// TwinCAT 3 PLC project PLC_Eksam2020ET_KEP
// ProgramVersion: 3.1.4023.0
// libraries:
//   Tc2_MC2, * (Beckhoff Automation GmbH)
//   Tc2_Standard, * (Beckhoff Automation GmbH)
//   Tc2_System, * (Beckhoff Automation GmbH)
//   Tc2_Utilities, * (Beckhoff Automation GmbH)
//   Tc3_Module, * (Beckhoff Automation GmbH)
//   SysTime,3.5.9.0,System
// project tree:
//   / Class Diagram.TcCD (not stored), GlobalTextList.TcGTLO, PlcTask.TcTTO, Visualization Manager.TcVMO (not stored)
//   GVLs/ FIO.TcGVL
//   POUs/ HMI.TcPOU, MAIN.TcPOU, P_5MovingToStack.TcPOU, P_3Pack.TcPOU, P_2PickUP.TcPOU, P_4Packing.TcPOU, P_6Stack.TcPOU, P_1Start.TcPOU
//   VISUs/ Visualization_Pos.TcVIS, Visualization_Start_Screen.TcVIS

CONFIGURATION PLC_Eksam2020ET_KEP
    RESOURCE PLC ON TwinCAT3
        TASK PlcTask(INTERVAL := T#10ms, PRIORITY := 20);
        PROGRAM MAIN WITH PlcTask : MAIN;
    END_RESOURCE
END_CONFIGURATION

// ---- GVLs/FIO.TcGVL
{attribute 'qualified_only'}
VAR_GLOBAL
	//SENSORS:


//Bool

bFACTORYRunning: BOOL;
bFACTORYPaused: BOOL;
bFACTORYReset1: BOOL;
bUnknown1: BOOL;
bUnknown2: BOOL;
bPP_ItemDetected: BOOL;
bPP_MovingX: BOOL;
bPP_MovingZ: BOOL;
bPP_BaseDetected: BOOL;
bPP_BaseClamped: BOOL;
bPP_PosLimitBase: BOOL;
bPP_LidClamped: BOOL;
bPP_PosLimitLid: BOOL;
bPP_PartLeaving: BOOL;
bPP_LidDetected: BOOL;
bEbStart: BOOL;
bEbReset: BOOL;
bEbStop: BOOL;
bEbES: BOOL;
bEbManual: BOOL;
bEbAuto: BOOL;
bSC_AtLeft: BOOL;
bInPaMovingXY: BOOL;
bInPaMovinZ: BOOL;
bInPaPosLimit: BOOL;
bInPaBoxDetected: BOOL;
bSC_AtMiddle: BOOL;
bSC_AtRight: BOOL;
bOutPaMovingXY: BOOL;
bOutPaMovingZ: BOOL;
bOutPaPosLimit: BOOL;
bOutPaBoxDetected: BOOL;
bSC_MovingZ: BOOL;
bSC_MovingX: BOOL;
bScAtLoad: BOOL;
bInPaSensBlue: BOOL;
bInPaSensGreen: BOOL;
bInPaSensMetal: BOOL;
bOutPaSens: BOOL;
bSsSensConv1: BOOL;
bSsSensConv2: BOOL;
bSsSensConv3: BOOL;
bPP_BaseSens: BOOL;


//Float

rFACTORYTimeScale: REAL;
rInPaPosY: LREAL;
rInPaPosZ: LREAL;
rInPaPosX: LREAL;
rOutPaPosY: REAL;
rOutPaPosZ: REAL;
rOutPaPosX: REAL;


//Int

iInVision: INT;
iRfidW_ReadData: INT;
iRfidW_CmdId: INT;
iRfidW_Status: INT;
iRfidR_ReadData: INT;
iRfidR_CmdId: INT;
iRfidR_Status: INT;

//ACTUATORS:

//Bool

bFACTORYRun: BOOL;
bFACTORYPause: BOOL;
bFACTORYReset2: BOOL;
bUnknown3: BOOL;
bUnknown4: BOOL;
bUnknown5: BOOL;
bUnknown6: BOOL;
bPP_Grab: BOOL;
bPP_MoveX: BOOL;
bPP_MoveZ: BOOL;
bInEmitBase: BOOL;
bPP_ConvLid: BOOL;
bPP_BaseClamp: BOOL;
bPP_PosRais_Base: BOOL;
bPP_LidClamp: BOOL;
bPP_PosRaise_Lid: BOOL;
bEbStartLight: BOOL;
bEbResetLight: BOOL;
bEbStopLight: BOOL;
bScConv1: BOOL;
bInConvGreen: BOOL;
bInConvMetal: BOOL;
bInConvSorting: BOOL;
bInConvBlue: BOOL;
bInPaGrab: BOOL;
bInPaToolRot: BOOL;
bSC_Left: BOOL;
bSC_Right: BOOL;
bSC_Lift: BOOL;
bOutPaGrab: BOOL;
bOutPaToolRot: BOOL;
bScConv2: BOOL;
bScLoadingConv: BOOL;
bInEmitMetalLid: BOOL;
bInEmitGreenLid: BOOL;
bInEmitBlueLid: BOOL;
bPP_ConvOut: BOOL;
bScEmitPallet: BOOL;
bRollerStopOut: BOOL;
bScConv3: BOOL;
bRfidW_ExeCmd: BOOL;
bRfidR_ExeCmd: BOOL;
bPP_ConvBase2: BOOL;
bPP_ConvBase1: BOOL;


//Float

rInPaMoveY: REAL;
rInPaMoveZ: REAL;
rInPaMoveX: REAL;
rOutPaMoveY: REAL;
rOutPaMoveZ: REAL;
rOutPaMoveX: REAL;

//Int

iFACTORYCameraPosition: INT;
iEbCounter: INT;
iSC_TargetPos: INT;
iRfidW_MemIndex: INT;
iRfidW_WriteData: INT;
iRfidW_Cmd: INT;
iRfidR_MemIndex: INT;
iRfidR_WriteData: INT;
iRfidR_Cmd: INT;
END_VAR

// ---- POUs/MAIN.TcPOU
PROGRAM MAIN
VAR
	
END_VAR

//In Main we just run all our program for pick and place stack mashine. 
//As you can see we have 6 program and a HMI program for our mashine. 

P_1Start();
P_2PickUP();
P_3Pack();
P_4Packing();
P_5MovingToStack();
P_6Stack();
HMI();

END_PROGRAM

// ---- POUs/P_1Start.TcPOU
PROGRAM P_1Start
VAR
	nState: INT;
	
END_VAR

VAR CONSTANT
	//Here we define our constant where we want the different positon to be. This is instead of making steps you can call this fixed steps.
	Standby    : INT := 00;
	Start		:INT := 01;
	atEntry    : INT := 10;
	Moving     : INT := 20;
	MovingStop : INT := 22;
	Waiting    : INT := 30;
	Stopping   : INT := 40;
	Resetting  : INT := 50;
	Estop      : INT := 99;
		
END_VAR

// This is our first program in the program we have made a state mashine  ( Case ... of ) to define what our system should do
// in the different states.



CASE nState OF
	Standby:		
		IF FIO.bEbStart=TRUE THEN
			FIO.bInEmitBase:=TRUE;
			nState:=Start;
		END_IF
		
	Start: // This is where we declair what should happen if a operator have turned the mashine in auto and pressed start.
			FIO.bInEmitBlueLid:=FALSE;
			FIO.bInEmitGreenLid:=FALSE;
			FIO.bInEmitMetalLid:=FALSE;
			
			
		IF FIO.bEbStart=TRUE AND FIO.bEbAuto=TRUE THEN 
			FIO.bInEmitBlueLid:=TRUE;     //Lids will start to spawn 
			FIO.bInEmitGreenLid:=TRUE;
			FIO.bInEmitMetalLid:=TRUE;
			nState:=Moving;
		END_IF

	Moving:	 //when the lids 
		IF FIO.bInEmitBlueLid=TRUE AND FIO.bInPaSensBlue=FALSE THEN
			FIO.bInConvBlue:=TRUE;       
		END_IF
		IF	FIO.bInEmitGreenLid=TRUE AND FIO.bInPaSensGreen=FALSE THEN
			FIO.bInConvGreen:=TRUE;
		END_IF
		IF FIO.bInEmitMetalLid=TRUE AND FIO.bInPaSensMetal=FALSE THEN
			FIO.bInConvMetal:=TRUE;
		END_IF	
			nState:=MovingStop;
			
	MovingStop:		
	 	IF FIO.bInPaSensBlue=TRUE THEN  
			FIO.bInConvBlue:=FALSE;
		END_IF
		IF FIO.bInPaSensGreen=TRUE THEN	
			FIO.bInConvGreen:=FALSE;
		END_IF	
		IF FIO.bInPaSensMetal=TRUE THEN	
			FIO.bInConvMetal:=FALSE;
		END_IF		
			nState := Waiting;			

		
//----------------------------------------------------------------------------//
	Waiting:
			nState:=Moving;
		
//----------------------------------------------------------------------------//
	Stopping:   //when stop is pressed we move into this statement the stop light turn on / This is also the state we start in when we turn on the PLC /System
		IF FIO.bEbStop = FALSE THEN
			FIO.bEbStopLight:=TRUE;
			FIO.bInEmitBase:=FALSE;
		ELSIF FIO.bEbReset=TRUE THEN
			FIO.bEbStopLight:=FALSE;
			nState:=Standby;	
		END_IF
//----------------------------------------------------------------------------//
			
			
		
//----------------------------------------------------------------------------// 			
	ELSE
			nState:=9999;				
END_CASE

IF NOT FIO.bEbStop THEN  
		nState:=Stopping;	
END_IF

END_PROGRAM

// ---- POUs/P_2PickUP.TcPOU
PROGRAM P_2PickUP
VAR
	nState: INT;
	
	//Vision Color for Lid
	Blue:	INT:=3;
	Green:	INT:=6;
	Metal:	INT:=9;
	
	//Timers for the different state to happen. It is good to put in timers so the machinery have time to do the different
	// state before it moves on to the next state else everything will happen really fast.
	fbTimerMoving : TON;	// Timer in the moving state so the XYZ arm have time to process before moving till next state.
	fbTimerPickUP : TON;	 // 
	fbTimerGrab : TON;
	fbTimerGrab2 : TON;
	fbTimerDrop : TON;
	fbTimerMovingLid : TON;
	fbTimerWaiting : TON;
END_VAR

VAR CONSTANT
	//This is the Constant Variables that we use to for the different state in our Case OF Statement.
	Standby: 		INT:=00;
	Start:			INT:=01;
	ReadVision: 	INT:=02;
	atEntry: 		INT:=10;
	Moving: 		INT:=20;
	PickUP:			INT:=21;
	PickUP2: 		INT:=22;
	Grab: 			INT:=23;
	Grab2: 			INT:=24;
	Drop: 			INT:=25;
	MovingLid: 		INT:=26;
	MovingLid2: 	INT:=27;
	MovingStop: 	INT:=29;
	Waiting: 		INT:=30;
	Stopping: 		INT:=40;
	Resetting: 		INT:=50;
	Estop:			INT:=99;
END_VAR

// This is our second program where we emit a base and let the vision cam tell us which color the base is so the first XYZ arm can pick up the lid and send if 
// to pack.


CASE nState OF 
	Standby:	
		IF FIO.bEbStart=TRUE THEN
			nState:=Start;
		END_IF	
	
	Start: 
			IF FIO.bInPaSensBlue AND FIO.bInPaSensGreen AND FIO.bInPaSensMetal THEN
				FIO.bInEmitBase:=TRUE;
				nState:=ReadVision;
			END_IF	
			
	ReadVision: //vision cam read the color of the base
				IF FIO.iInVision=Blue THEN
					FIO.rInPaMoveX:=9;			
					nState:=Moving;	
				END_IF
				IF FIO.iInVision=Green THEN
					FIO.rInPaMoveX:=5;					
					nState:=Moving;
				END_IF
				IF FIO.iInVision=Metal THEN 
					FIO.rInPaMoveX:=1;			
					nState:=Moving;
				END_IF
				
	Moving:
		IF FIO.rInPaMoveX=9 OR FIO.rInPaMoveX=5 OR FIO.rInPaMoveX=1 THEN
			FIO.rInPaMoveY:=0.5;
		 fbTimerMoving(IN:=TRUE,PT:=T#1S);
		 IF fbTimerMoving.Q THEN
			fbTimerMoving(IN:=FALSE);
			nState:=PickUP; 
		 END_IF		
		END_IF
	
	PickUP:
		IF FIO.rInPaMoveY=0.5 THEN
			FIO.rInPaMoveZ:=9;
			FIO.bInPaToolRot:=TRUE;
			fbTimerPickUP(IN:=TRUE,PT:=T#1S);
		 IF fbTimerPickUP.Q THEN
			 fbTimerPickUP(IN:=FALSE);
			nState:=Grab; 
		 END_IF	
		END_IF
		
	Grab:
		IF FIO.rInPaMoveZ=9 THEN
			FIO.bInPaGrab:=TRUE;
		fbTimerGrab(IN:=TRUE,PT:=T#1S);
		 IF fbTimerGrab.Q THEN
			fbTimerGrab(IN:=FALSE);
			nState:=Grab2; 
		 END_IF
		END_IF
		
	Grab2:	
		IF FIO.bInPaGrab=TRUE THEN
			FIO.rInPaMoveZ:=5;
			FIO.rInPaMoveY:=8;
			fbTimerGrab2(IN:=TRUE,PT:=T#1S);	
			IF fbTimerGrab2.Q THEN
				fbTimerGrab2(IN:=FALSE);
				nState:=Drop;
		 	END_IF				
		END_IF
	
	Drop:
		IF FIO.bInPaGrab=TRUE THEN
			FIO.rInPaMoveZ:=8.5;
			fbTimerDrop(IN:=TRUE,PT:=T#1S);	
			IF fbTimerDrop.Q THEN
				fbTimerDrop(IN:=FALSE);
				nState:=MovingLid; 
		 	END_IF
		 END_IF
		 
	MovingLid:				
			IF FIO.rInPaMoveZ=8.5 THEN
				FIO.bInPaGrab:=FALSE;
			END_IF
				fbTimerMovingLid(IN:=TRUE,PT:=T#1S);	
			IF fbTimerMovingLid.Q THEN
				fbTimerMovingLid(IN:=FALSE);
				nState:=MovingLid2; 
		 	END_IF
			
	MovingLid2:		
			IF FIO.bInPaGrab=FALSE THEN
				FIO.rInPaMoveX:=0;
				FIO.rInPaMoveY:=0;
				FIO.rInPaMoveZ:=0;
				FIO.bInPaToolRot:=FALSE;
				FIO.bInConvSorting:=TRUE;
				nState:=waiting; 	
			END_IF
//----------------------------------------------------------------------------//
	Waiting:
			IF FIO.bPP_LidClamp=TRUE THEN
			fbTimerWaiting(IN:=TRUE,PT:=T#1S);	
			IF fbTimerWaiting.Q THEN
				fbTimerWaiting(IN:=FALSE); 
				nState:=Start;
			END_IF
			END_IF
//----------------------------------------------------------------------------//

		

	
	Stopping:
		IF FIO.bEbStop = FALSE THEN
			FIO.bEbStopLight:=TRUE;
		ELSIF FIO.bEbReset=TRUE THEN
				FIO.bEbStopLight:=FALSE;	
			nState:=Standby;	
		END_IF	

//----------------------------------------------------------------------------// 
	ELSE
		nState:=9999;	
END_CASE

IF NOT FIO.bEbStop THEN
		nState:=Stopping;	
END_IF

END_PROGRAM

// ---- POUs/P_3Pack.TcPOU
PROGRAM P_3Pack
VAR
	nState: INT;
	
	fbTimerConvs: TON;
	fbTimerPickUP: TON;
	fbTimerGrab: TON;
	fbMyTimer4: TON;
	fbMyTimer5: TON;
	fbMyTimer6: TON;
	fbMyTimer7 : TON;
	fbMyTimer8 : TON;
	fbMyTimer9 : TON;
	F_TRIGLid:F_TRIG;
END_VAR

VAR CONSTANT
	Standby: 	INT:=00;
	Start:		INT:=01;
	atEntry: 	INT:=10;
	Moving: 	INT:=20;
	MovingStopLidClamp: INT:=21;
	MovingStopBase: 	INT:=22;
	PickUP: 	INT:=23;
	PickUP2: 	INT:=24;
	Grab: 		INT:=25;
	Grab2: 		INT:=26;
	Drop: 		INT:=27;
	Moving2: 	INT:=28;
	MovingPack: INT:=29;
	RaiseBase:	INT:=65;
	StoppingAtSens: INT:= 67;
	Stopping: 	INT:=40;
	Resetting: 	INT:=50;
	Clamp:		INT:=60;
	Waiting: 	INT:=30;
	Estop: 		INT:=99;
	
	
END_VAR

// This is our third program  in this program we put the lid together with the base so it can be a box.


F_TRIGLid(CLK:=FIO.bPP_LidDetected);  //trigger for the sense at the lid pack

CASE nState OF
	Standby: 
		nState:=Start;
 
	Start:    
		IF FIO.bInConvSorting=TRUE THEN
			FIO.bPP_ConvBase1:=TRUE;
			FIO.bPP_ConvBase2:=TRUE;
			FIO.bPP_ConvLid:=TRUE;
			fbTimerConvs(IN:=TRUE,PT:=T#1S);
			IF fbTimerConvs.Q THEN
			fbTimerConvs(IN:=FALSE); 
			nState:=MovingStopBase;
		END_IF	
	END_IF
	
	MovingStopBase:
			IF FIO.bPP_BaseDetected=TRUE THEN
				FIO.bPP_ConvBase1:=FALSE;						
				nState:=MovingStopLidClamp;			
			END_IF
	
			
	MovingStopLidClamp:	  // where the clam for lid and base are activated.
		IF F_TRIGLid.Q THEN
			FIO.bPP_LidClamp:=TRUE;
			FIO.bPP_BaseClamp:=TRUE;	
			nState:=PickUP;
		END_IF
		
	PickUP:
		IF FIO.bPP_LidClamp=TRUE AND FIO.bPP_BaseClamp=TRUE THEN
			FIO.bPP_ConvBase2:=FALSE;
			FIO.bInConvSorting:=FALSE;
			FIO.bPP_MoveX:=TRUE;
			fbTimerPickUP(IN:=TRUE,PT:=T#2S);
				IF fbTimerPickUP.Q THEN
					fbTimerPickUP(IN:=FALSE); 
					nState:=Grab;
				END_IF
		END_IF
	
	Grab:
		IF FIO.bPP_MoveX=TRUE THEN
			FIO.bPP_ConvLid:=FALSE;
			FIO.bPP_MoveZ:=TRUE;
			FIO.bPP_Grab:=TRUE;
			fbTimerGrab(IN:=TRUE,PT:=T#2S);
				IF fbTimerGrab.Q THEN
					fbTimerGrab(IN:=FALSE);
					FIO.bPP_LidClamp:=FALSE; 
					nState:=Grab2;
				END_IF
		END_IF

	Grab2:
		IF FIO.bPP_Grab=TRUE THEN
			FIO.bPP_MoveZ:=FALSE;
			fbMyTimer4(IN:=TRUE,PT:=T#2S);
				IF fbMyTimer4.Q THEN
					fbMyTimer4(IN:=FALSE); 
					FIO.bPP_MoveX:=FALSE;
					nState:=Drop;	
				END_IF			
		END_IF	
	
	Drop:
		IF FIO.bPP_MoveX=FALSE THEN
		fbMyTimer5(IN:=TRUE,PT:=T#2S);
			IF fbMyTimer5.Q THEN
				fbMyTimer5(IN:=FALSE); 
				FIO.bPP_MoveZ:=TRUE;
				nState:=Moving2;	
			END_IF	
		END_IF		
	
	Moving2:
		IF FIO.bPP_MovingX=FALSE THEN	
		fbMyTimer6(IN:=TRUE,PT:=T#2S);
			IF fbMyTimer6.Q THEN
				fbMyTimer6(IN:=FALSE);
				FIO.bPP_Grab:=FALSE; 
				nState:=MovingPack;	
			END_IF							
		END_IF
	
	MovingPack:
		IF FIO.bPP_Grab=FALSE THEN
			FIO.bPP_MoveZ:=FALSE;
			FIO.bPP_BaseClamp:=FALSE;
			fbMyTimer7(IN:=TRUE,PT:=T#2S);
			IF fbMyTimer7.Q THEN
				fbMyTimer7(IN:=FALSE);
				nState:=RaiseBase;	
			END_IF	
		END_IF
	
	RaiseBase:
		IF FIO.bPP_MoveZ=FALSE THEN
			FIO.bPP_PosRais_Base:=TRUE;
			FIO.bPP_ConvBase2:=TRUE;
			FIO.bPP_ConvOut:=TRUE;
			fbMyTimer8(IN:=TRUE,PT:=T#2S);
			IF fbMyTimer8.Q THEN
				fbMyTimer8(IN:=FALSE);
				FIO.bPP_PosRais_Base:=FALSE;
				nState:=StoppingAtSens;	
			END_IF	
		END_IF
		
	StoppingAtSens:
		IF FIO.bOutPaSens = TRUE THEN
			FIO.bPP_ConvOut:=FALSE;
			nState:=Waiting;
		END_IF
//----------------------------------------------------------------------------//

	Waiting:
			nState:=Standby;
		
//----------------------------------------------------------------------------//		
		
	ELSE
		nState:=9999;	
END_CASE

END_PROGRAM

// ---- POUs/P_4Packing.TcPOU
PROGRAM P_4Packing
VAR
	nState: INT;
	
	//Timers
	fbTimerGrabX : TON;
	fbTimerGrabY : TON;
	fbTimerGrabZ : TON;
	fbTimerGrab : TON;
	fbTimerLift : TON;
	fbTimerDrop1 : TON;
	fbTimerDrop2 : TON;
	fbTimerMoving2 : TON;
	fbTimerMoving3 : TON;
	fbTimerMovingLoad : TON;
	fbTimerWaiting : TON;
	fbTimerEmitPal: TON;
	
	iCounterTrig: R_trig;
	
END_VAR
VAR CONSTANT
	//Here we define our constant where we want the different positon to be. This is instead of making steps you can call this fixed steps.
	Standby: 	INT:=00;
	GrabX:		INT:=10;
	GrabY:		INT:=11;
	GrabZ:		INT:=12;
	Grab:		INT:=13;
	Lift:		INT:=15;
	Drop1:		INT:=20;
	Drop2:		INT:=21;
	Moving1    : INT := 30;
	Moving2    : INT := 31;
	Moving3    : INT := 32;
	MovingStop : INT := 22;
	AtLoad:		INT:=35;	
	Waiting    : INT := 40;
	Stopping   : INT := 50;
	Resetting  : INT := 60;
	Estop      : INT := 99;
		
END_VAR

// This is our fourth program is where we count the anount of boxes that have been put together  and the second xyz arm will pick up the box 
// and place it on the pallet.

iCounterTrig(CLK:=FIO.bPP_PosRais_Base);  //define a trigger so we can use it to count the amount of boxes that have been put together.  

IF iCounterTrig.Q THEN                    //box counter
	FIO.iEbCounter:=FIO.iEbCounter+1;
END_IF


 
CASE nState OF
	
	Standby:      //the sensor is true when there are a box and a palled will emit 
		IF  FIO.bOutPaSens=TRUE THEN
			FIO.bScEmitPallet:=TRUE;	
			nState:=GrabX;		
		END_IF	
				

	GrabX:		//we move the XYZ arm in the X position 
		IF FIO.bOutPaSens=TRUE THEN    
			FIO.rOutPaMoveX:=4.5;
			fbTimerGrabX(IN:=TRUE,PT:=T#1S);	
			IF fbTimerGrabX.Q THEN
				fbTimerGrabX(IN:=FALSE); 
				nState:=GrabY;
			END_IF	
		END_IF

	GrabY:	//we move the XYZ arm in the Y position 
		IF FIO.rOutPaMoveX=4.5 THEN 
			FIO.rOutPaMoveY:=9.5;
			fbTimerGrabY(IN:=TRUE,PT:=T#1S);	
			IF fbTimerGrabY.Q THEN
				fbTimerGrabY(IN:=FALSE); 
				nState:=GrabZ;
			END_IF	
		END_IF
	
	GrabZ:  //we move the XYZ arm in the Z position 
		IF FIO.rOutPaMoveY=9.5 THEN 
			FIO.rOutPaMoveZ:=8.5;
			FIO.bOutPaToolRot:=TRUE;
			fbTimerGrabZ(IN:=TRUE,PT:=T#2S);	
			IF fbTimerGrabZ.Q THEN
				fbTimerGrabZ(IN:=FALSE); 
				nState:=Grab;
			END_IF				
		END_IF
	
	Grab:   //we here we turn the grab on so it can pick up a box
		IF FIO.bOutPaBoxDetected=TRUE THEN
			FIO.bOutPaGrab:=TRUE;
			fbTimerGrab(IN:=TRUE,PT:=T#1S);
			 IF fbTimerGrab.Q THEN
				fbTimerGrab(IN:=FALSE);
				nState:=Lift; 
		 	END_IF
		END_IF	
		
	Lift:    //here we lift the box
		IF FIO.bOutPaGrab=TRUE THEN
			FIO.rOutPaMoveZ:=0;
			fbTimerLift(IN:=TRUE,PT:=T#1S);
			 IF fbTimerLift.Q THEN
				fbTimerLift(IN:=FALSE);
				nState:=Drop1;
		 	END_IF					
		END_IF	

	Drop1:  // here move in Y axes so it is almost in the middle of the pallet
		IF FIO.rOutPaMoveZ=0 THEN
			FIO.rOutPaMoveY:=1.5;
			fbTimerDrop1(IN:=TRUE,PT:=T#1S);
			 IF fbTimerDrop1.Q THEN
				fbTimerDrop1(IN:=FALSE);
				nState:=Drop2;
		 	END_IF
		END_IF	
		
	Drop2:  //here we move the arm in Z position where we lower the har closer to the pallet and then we drop the box
		IF FIO.bOutPaGrab=TRUE THEN
			FIO.rOutPaMoveZ:=10;
			fbTimerDrop2(IN:=TRUE,PT:=T#1S);
			 IF fbTimerDrop2.Q THEN
				fbTimerDrop2(IN:=FALSE);
				FIO.bOutPaGrab:=FALSE;
				nState:=Waiting;;
		 	END_IF	
		END_IF


		
//----------------------------------------------------------------------------//

	Waiting:
			nState:=Standby;
		
			
		
//----------------------------------------------------------------------------//


	ELSE
		nState:=9999;	
END_CASE

END_PROGRAM

// ---- POUs/P_5MovingToStack.TcPOU
PROGRAM P_5MovingToStack
VAR
	nState: INT;
	
	//Timers
	fbTimerGrabX : TON;
	fbTimerGrabY : TON;
	fbTimerGrabZ : TON;
	fbTimerGrab : TON;
	fbTimerLift : TON;
	fbTimerDrop1 : TON;
	fbTimerDrop2 : TON;
	fbTimerMoving1 : TON;
	fbTimerMoving2 : TON;
	fbTimerMoving3 : TON;
	fbTimerMovingLoad : TON;
	fbTimerWaiting : TON;
	fbTimerEmitPal: TON;
END_VAR
VAR CONSTANT
	Standby: 	INT := 00;
	atEntry: 	INT := 10;
	GrabX:		INT:=10;
	GrabY:		INT:=11;
	GrabZ:		INT:=12;
	Grab:		INT:=13;
	Lift:		INT:=15;
	Drop1:		INT:=20;
	Drop2:		INT:=21;
	Moving1    : INT := 30;
	Moving2    : INT := 31;
	Moving3    : INT := 32;
	MovingStop : INT := 22;
	AtLoad:		INT:=35;	
	Waiting    : INT := 40;
	Stopping   : INT := 50;
	Resetting  : INT := 60;
	Estop      : INT := 9999;
	
	
END_VAR

// This is our fifth program where we make sure to emit a pallet sent the XYZ arn to it's start position. 
// it is also here where we move the pallet with box so it can be stacked in the next program

//we have a If statement when the sensor at the OutPaSens is true then we emit a pallet else we don't.
IF  FIO.bOutPaSens=TRUE THEN    
	FIO.bScEmitPallet:=TRUE;
ELSE 
	FIO.bScEmitPallet:=FALSE;			
END_IF	

CASE nState OF 
	Standby: // we make sure that the grab have stop and there are no box at the OutPaSens then the xyz arm cna move to its home position. 
		IF FIO.bOutPaGrab=FALSE AND FIO.bSsSensConv1=TRUE AND FIO.bOutPaSens=FALSE THEN
			FIO.rOutPaMoveX:=0;
			FIO.rOutPaMoveY:=0;
			FIO.rOutPaMoveZ:=0;
			FIO.bOutPaToolRot:=FALSE;
			fbTimerMoving2(IN:=TRUE,PT:=T#1S);
			IF fbTimerMoving2.Q THEN
				fbTimerMoving2(IN:=FALSE);
				nState:=Moving1;
			END_IF
		END_IF
		
	Moving1:  // if the Sensor at Conveyor1 is True it means there is a pallet  and the grab is false that mean that the box have been delivered 
			IF FIO.bSsSensConv1=TRUE AND FIO.bOutPaGrab=FALSE AND FIO.rOutPaMoveX=0 THEN  
					FIO.bScConv1:=TRUE; //here we start the convayer so the pallet can move 
					nState:=Moving2;
			END_IF

	
	Moving2:  // moving to next conveayer 
		IF FIO.bSsSensConv2=TRUE THEN
			FIO.bScConv2:=TRUE;
			fbTimerMoving2(IN:=TRUE,PT:=T#1S);
			 IF fbTimerMoving2.Q THEN
				fbTimerMoving2(IN:=FALSE);
				FIO.bScConv1:=FALSE;
				nState:=Moving3;
		 	END_IF					 
		END_IF
	
	Moving3: //moving though the last conveyor before it is at the load conveyor. 
		IF FIO.bSsSensConv3=TRUE THEN 
			FIO.bScConv3:=TRUE;
			fbTimerMoving3(IN:=TRUE,PT:=T#1S);
			 IF fbTimerMoving3.Q THEN
				fbTimerMoving3(IN:=FALSE);
				FIO.bScConv2:=FALSE;
				nState:=Waiting;
		 	END_IF						
		END_IF
		
//----------------------------------------------------------------------------//

	Waiting:
			nState:=Standby;
		
//----------------------------------------------------------------------------//		
		
	ELSE 
		nState:=9999; 	
		
END_CASE

END_PROGRAM

// ---- POUs/P_6Stack.TcPOU
PROGRAM P_6Stack
VAR
	nState: INT;
	
	//Timers
	fbTimerMovingLoad: TON;
	fbTimerLift: TON;
	fbTimerToSpace: TON;
	fbTimerPlace: TON;
	fbTimerCounter: TON;
	fbTimerHoming: TON;
	
	
	AtLoadTrig:R_TRIG;		

	//INT
	nCounter         : INT := 0;
END_VAR

VAR CONSTANT
	//Here we define our constant where we want the different positon to be. This is instead of making steps you can call this fixed steps.
	Start		:INT:=00;
	AtLoad		:INT:=01;
	PickUP 		:INT := 02;
	LiftPallet         : INT := 03;
	RetractForksLeft   : INT := 04;
	MovingToSpace      : INT := 05;
	DeliverPart        : INT := 06;
	PlacePallet        : INT := 07;
	RetractRight       : INT := 08;
	Homing             : INT := 09;
	Retry   		   : INT := 10;
	Moving     : INT := 20;
	MovingStop : INT := 22;
	GetPart            : INT := 50;
	GetPartPick        : INT := 51;
	PartPickUp    	   : INT := 52;
	PickUpPart         : INT := 53;
	PartPicked 		   : INT := 54;
	MoveToUnload       : INT := 55;
	UnloadPart 		   : INT := 56;
	PlacePart          : INT := 57;
	Waiting    : INT := 30;	
	Stopping   : INT := 40;
	Resetting  : INT := 60;
	Estop      : INT := 9999;		
END_VAR

// This is our sixth program the stacker robot will pick up the pallet at load and stack them into the different shelf from 1 to 54. 


AtLoadTrig(CLK:=FIO.bScAtLoad);


CASE nState OF
		Start: //Entry of the Palled 
			IF FIO.bScAtLoad=FALSE AND FIO.bScConv3=TRUE THEN
				FIO.bScLoadingConv:=TRUE;                       //turning on the load conveyor
			END_IF
				FIO.iSC_TargetPos := 21474; //This is the value that sends the crane home.
			
			IF AtLoadTrig.Q THEN // counter for the stack robot to know which shelf to put the palled in shelf no = anount of pallet that have been at entry.
			nCounter:=nCounter+1;
			END_IF
			IF FIO.bScAtLoad=TRUE THEN
				nState := AtLoad;
			END_IF
		
		AtLoad:	 // Pallet is at load, the different conveyor will go false when pallet is at load.
		IF FIO.bScAtLoad=TRUE THEN 
			FIO.bScLoadingConv:=FALSE;
			fbTimerMovingLoad(IN:=TRUE,PT:=T#1S);
			IF fbTimerMovingLoad.Q THEN
				fbTimerMovingLoad(IN:=FALSE);
				FIO.bScConv3:=FALSE;
				nState := PickUP;
		 	END_IF						
		END_IF	

	PickUP:  // here we make sure that the the stack robot are at home and there pallet at the load and moving x and z are false before it cna pick up a pallet.
		IF FIO.bScAtLoad=TRUE AND FIO.iSC_TargetPos = 21474 AND FIO.bSC_MovingX=FALSE and FIO.bSC_MovingZ=FALSE THEN
			FIO.bSc_Left := TRUE;
			nState := LiftPallet;
		END_IF
	
	LiftPallet:	 // there the pallet gets picked up	
		IF FIO.bSc_AtLeft=TRUE THEN
			FIO.bSc_Lift:=TRUE;
			fbTimerLift(IN:=TRUE,PT:=T#1S);	
			IF fbTimerLift.Q THEN
				fbTimerLift(IN:=FALSE);
				FIO.bSc_Left :=FALSE; 
				nState := RetractForksLeft;
			END_IF	
		END_IF
	
	RetractForksLeft:  // here er made an extra step to give time for the fock to come back before we move to the next state
			nState:= MovingToSpace;
			
	MovingToSpace:	// here we make sure that the pallet are at mid before the stack robot moves again and we cound which palle 
		IF 	FIO.bSC_AtMiddle=TRUE THEN
			FIO.iSC_TargetPos:=nCounter;    //here we set the pallet count = the target pos which is the space in the shelf
			fbTimerToSpace(IN:=TRUE,PT:=T#2S);	
			IF fbTimerToSpace.Q THEN
				fbTimerToSpace(IN:=FALSE);
				nState := DeliverPart;
			END_IF
		END_IF

	DeliverPart: // here we put pallet into shelf                             
		IF FIO.bSC_MovingX=FALSE THEN
		FIO.bSc_Right := TRUE;                    
		nState := PlacePallet;
		END_IF
		
	PlacePallet:   
		IF FIO.bSc_AtRight=TRUE THEN
			FIO.bSc_Lift:=FALSE;
			fbTimerPlace(IN:=TRUE,PT:=T#1S);	
			IF fbTimerPlace.Q THEN
				fbTimerPlace(IN:=FALSE);
				nState := RetractRight;
			END_IF	
		END_IF

   		RetractRight:   //retract the arm     
		    IF FIO.bSc_Lift=FALSE THEN
				FIO.bSc_Right:=FALSE;
			fbTimerHoming(IN:=TRUE,PT:=T#1S);	
			IF fbTimerHoming.Q THEN
				fbTimerHoming(IN:=FALSE);
				nState := Homing; 		
			END_IF				
		END_IF

	Homing:		//moving to homing
		IF FIO.bSc_AtMiddle=TRUE THEN
			FIO.iSc_TargetPos := 21474;
			nState := Start;	
		END_IF		
		
	ELSE

	nState:=9999;		
	
END_CASE

END_PROGRAM

// ---- POUs/HMI.TcPOU
PROGRAM HMI
VAR

	SpaceOcc1: BOOL;
	
	nState: INT;
	nLastState: INT;
	
	nCounter: INT;
	EmitTrig:R_TRIG;

	Lamp1_Blue: BOOL;
	Lamp1_Green: BOOL;
	Lamp1_Metal: BOOL;	
	Lamp2_Blue: BOOL;
	Lamp2_Green: BOOL;
	Lamp2_Metal: BOOL;
	Lamp3_Blue: BOOL;
	Lamp3_Green: BOOL;
	Lamp3_Metal: BOOL;
	Lamp4_Blue: BOOL;
	Lamp4_Green: BOOL;
	Lamp4_Metal: BOOL;
	Lamp5_Blue: BOOL;
	Lamp5_Green: BOOL;
	Lamp5_Metal: BOOL;
	Lamp6_Blue: BOOL;
	Lamp6_Green: BOOL;
	Lamp6_Metal: BOOL;
	Lamp7_Blue: BOOL;
	Lamp7_Green: BOOL;
	Lamp7_Metal: BOOL;	
	Lamp8_Blue: BOOL;
	Lamp8_Green: BOOL;
	Lamp8_Metal: BOOL;
	Lamp9_Blue: BOOL;
	Lamp9_Green: BOOL;
	Lamp9_Metal: BOOL;
	Lamp10_Blue: BOOL;
	Lamp10_Green: BOOL;
	Lamp10_Metal: BOOL;
	Lamp11_Blue: BOOL;
	Lamp11_Green: BOOL;
	Lamp11_Metal: BOOL;
	Lamp12_Blue: BOOL;
	Lamp12_Green: BOOL;
	Lamp12_Metal: BOOL;
	Lamp13_Blue: BOOL;
	Lamp13_Green: BOOL;
	Lamp13_Metal: BOOL;
	Lamp14_Blue: BOOL;
	Lamp14_Green: BOOL;
	Lamp14_Metal: BOOL;
	Lamp15_Blue: BOOL;
	Lamp15_Green: BOOL;
	Lamp15_Metal: BOOL;
	Lamp16_Blue: BOOL;
	Lamp16_Green: BOOL;
	Lamp16_Metal: BOOL;
	Lamp17_Blue: BOOL;
	Lamp17_Green: BOOL;
	Lamp17_Metal: BOOL;
	Lamp18_Blue: BOOL;
	Lamp18_Green: BOOL;
	Lamp18_Metal: BOOL;
	Lamp19_Blue: BOOL;
	Lamp19_Green: BOOL;
	Lamp19_Metal: BOOL;	
	Lamp20_Blue: BOOL;
	Lamp20_Green: BOOL;
	Lamp20_Metal: BOOL;
	Lamp21_Blue: BOOL;
	Lamp21_Green: BOOL;
	Lamp21_Metal: BOOL;
	Lamp22_Blue: BOOL;
	Lamp22_Green: BOOL;
	Lamp22_Metal: BOOL;
	Lamp23_Blue: BOOL;
	Lamp23_Green: BOOL;
	Lamp23_Metal: BOOL;
	Lamp24_Blue: BOOL;
	Lamp24_Green: BOOL;
	Lamp24_Metal: BOOL;
	Lamp25_Blue: BOOL;
	Lamp25_Green: BOOL;
	Lamp25_Metal: BOOL;
	Lamp26_Blue: BOOL;
	Lamp26_Green: BOOL;
	Lamp26_Metal: BOOL;
	Lamp27_Blue: BOOL;
	Lamp27_Green: BOOL;
	Lamp27_Metal: BOOL;
	Lamp28_Blue: BOOL;
	Lamp28_Green: BOOL;
	Lamp28_Metal: BOOL;
	Lamp29_Blue: BOOL;
	Lamp29_Green: BOOL;
	Lamp29_Metal: BOOL;	
	Lamp30_Blue: BOOL;
	Lamp30_Green: BOOL;
	Lamp30_Metal: BOOL;
	Lamp31_Blue: BOOL;
	Lamp31_Green: BOOL;
	Lamp31_Metal: BOOL;
	Lamp32_Blue: BOOL;
	Lamp32_Green: BOOL;
	Lamp32_Metal: BOOL;
	Lamp33_Blue: BOOL;
	Lamp33_Green: BOOL;
	Lamp33_Metal: BOOL;
	Lamp34_Blue: BOOL;
	Lamp34_Green: BOOL;
	Lamp34_Metal: BOOL;
	Lamp35_Blue: BOOL;
	Lamp35_Green: BOOL;
	Lamp35_Metal: BOOL;
	Lamp36_Blue: BOOL;
	Lamp36_Green: BOOL;
	Lamp36_Metal: BOOL;
	Lamp37_Blue: BOOL;
	Lamp37_Green: BOOL;
	Lamp37_Metal: BOOL;
	Lamp38_Blue: BOOL;
	Lamp38_Green: BOOL;
	Lamp38_Metal: BOOL;
	Lamp39_Blue: BOOL;
	Lamp39_Green: BOOL;
	Lamp39_Metal: BOOL;	
	Lamp40_Blue: BOOL;
	Lamp40_Green: BOOL;
	Lamp40_Metal: BOOL;	
	Lamp41_Blue: BOOL;
	Lamp41_Green: BOOL;
	Lamp41_Metal: BOOL;	
	Lamp42_Blue: BOOL;
	Lamp42_Green: BOOL;
	Lamp42_Metal: BOOL;	
	Lamp43_Blue: BOOL;
	Lamp43_Green: BOOL;
	Lamp43_Metal: BOOL;	
	Lamp44_Blue: BOOL;
	Lamp44_Green: BOOL;
	Lamp44_Metal: BOOL;	
	Lamp45_Blue: BOOL;
	Lamp45_Green: BOOL;
	Lamp45_Metal: BOOL;	
	Lamp46_Blue: BOOL;
	Lamp46_Green: BOOL;
	Lamp46_Metal: BOOL;	
	Lamp47_Blue: BOOL;
	Lamp47_Green: BOOL;
	Lamp47_Metal: BOOL;	
	Lamp48_Blue: BOOL;
	Lamp48_Green: BOOL;
	Lamp48_Metal: BOOL;	
	Lamp49_Blue: BOOL;
	Lamp49_Green: BOOL;
	Lamp49_Metal: BOOL;		
	Lamp50_Blue: BOOL;
	Lamp50_Green: BOOL;
	Lamp50_Metal: BOOL;	
	Lamp51_Blue: BOOL;
	Lamp51_Green: BOOL;
	Lamp51_Metal: BOOL;	
	Lamp52_Blue: BOOL;
	Lamp52_Green: BOOL;
	Lamp52_Metal: BOOL;	
	Lamp53_Blue: BOOL;
	Lamp53_Green: BOOL;
	Lamp53_Metal: BOOL;	
	Lamp54_Blue: BOOL;
	Lamp54_Green: BOOL;
	Lamp54_Metal: BOOL;		



END_VAR

// In this program we setup the link between the stacking shelf with the HMI,
// it is here we set the lamps that will show what color box that are on the shelf
// and what shelf number the boxes are on. 
// It is also here we link the start and stop from HMI, and the auto status. 
// We have not made so you can put the system in auto on the HMI, this is due to safty. 

EmitTrig(CLK:=FIO.bPP_BaseSens);

IF EmitTrig.Q THEN				// This is the counter that are linked with the HIM to se the shelf number the boxes go in.
	nCounter:=nCounter+1;
END_IF


//---------------------------------------------------

IF nCounter = 1 AND FIO.iInVision = 3 THEN   // Linking the self number with the color of the box  throw the vision sencor.
        Lamp1_Blue := TRUE;
END_IF	
IF nCounter = 1 AND FIO.iInVision = 6 THEN  
        Lamp1_Green := TRUE;
END_IF		
IF nCounter = 1 AND FIO.iInVision = 9 THEN
        Lamp1_Metal := TRUE;
END_IF		

//---------------------------------------------------
	
IF nCounter = 2 AND FIO.iInVision = 3 THEN
        Lamp2_Blue := TRUE;
END_IF	
IF nCounter = 2 AND FIO.iInVision = 6 THEN
        Lamp2_Green := TRUE;
END_IF		
IF nCounter = 2 AND FIO.iInVision = 9 THEN
        Lamp2_Metal := TRUE;
END_IF	


//---------------------------------------------------

IF nCounter = 3 AND FIO.iInVision = 3 THEN
        Lamp3_Blue := TRUE;
END_IF	
IF nCounter = 3 AND FIO.iInVision = 6 THEN
        Lamp3_Green := TRUE;
END_IF		
IF nCounter = 3 AND FIO.iInVision = 9 THEN
        Lamp3_Metal := TRUE;
END_IF


//---------------------------------------------------

IF nCounter = 4 AND FIO.iInVision = 3 THEN
        Lamp4_Blue := TRUE;
END_IF	
IF nCounter = 4 AND FIO.iInVision = 6 THEN
        Lamp4_Green := TRUE;
END_IF		
IF nCounter = 4 AND FIO.iInVision = 9 THEN
        Lamp4_Metal := TRUE;
END_IF

//---------------------------------------------------

IF nCounter = 5 AND FIO.iInVision = 3 THEN
        Lamp5_Blue := TRUE;
END_IF	
IF nCounter = 5 AND FIO.iInVision = 6 THEN
        Lamp5_Green := TRUE;
END_IF		
IF nCounter = 5 AND FIO.iInVision = 9 THEN
        Lamp5_Metal := TRUE;
END_IF

//---------------------------------------------------

IF nCounter = 6 AND FIO.iInVision = 3 THEN
        Lamp6_Blue := TRUE;
END_IF	
IF nCounter = 6 AND FIO.iInVision = 6 THEN
        Lamp6_Green := TRUE;
END_IF		
IF nCounter = 6 AND FIO.iInVision = 9 THEN
        Lamp6_Metal := TRUE;
END_IF

//---------------------------------------------------

IF nCounter = 7 AND FIO.iInVision = 3 THEN
        Lamp7_Blue := TRUE;
END_IF	
IF nCounter = 7 AND FIO.iInVision = 6 THEN
        Lamp7_Green := TRUE;
END_IF		
IF nCounter = 7 AND FIO.iInVision = 9 THEN
        Lamp7_Metal := TRUE;
END_IF

//---------------------------------------------------

IF nCounter = 8 AND FIO.iInVision = 3 THEN
        Lamp8_Blue := TRUE;
END_IF	
IF nCounter = 8 AND FIO.iInVision = 6 THEN
        Lamp8_Green := TRUE;
END_IF		
IF nCounter = 8 AND FIO.iInVision = 9 THEN
        Lamp8_Metal := TRUE;
END_IF

//---------------------------------------------------

IF nCounter = 9 AND FIO.iInVision = 3 THEN
        Lamp9_Blue := TRUE;
END_IF	
IF nCounter = 9 AND FIO.iInVision = 6 THEN
        Lamp9_Green := TRUE;
END_IF		
IF nCounter = 9 AND FIO.iInVision = 9 THEN
        Lamp9_Metal := TRUE;
END_IF

//---------------------------------------------------

IF nCounter = 10 AND FIO.iInVision = 3 THEN
        Lamp10_Blue := TRUE;
END_IF	
IF nCounter = 10 AND FIO.iInVision = 6 THEN
        Lamp10_Green := TRUE;
END_IF		
IF nCounter = 10 AND FIO.iInVision = 9 THEN
        Lamp10_Metal := TRUE;
END_IF

//---------------------------------------------------

IF nCounter = 11 AND FIO.iInVision = 3 THEN
        Lamp11_Blue := TRUE;
END_IF	
IF nCounter = 11 AND FIO.iInVision = 6 THEN
        Lamp11_Green := TRUE;
END_IF		
IF nCounter = 11 AND FIO.iInVision = 9 THEN
        Lamp11_Metal := TRUE;
END_IF

//---------------------------------------------------

IF nCounter = 12 AND FIO.iInVision = 3 THEN
        Lamp12_Blue := TRUE;
END_IF	
IF nCounter = 12 AND FIO.iInVision = 6 THEN
        Lamp12_Green := TRUE;
END_IF		
IF nCounter = 12 AND FIO.iInVision = 9 THEN
        Lamp12_Metal := TRUE;
END_IF

//---------------------------------------------------

IF nCounter = 13 AND FIO.iInVision = 3 THEN
        Lamp13_Blue := TRUE;
END_IF	
IF nCounter = 13 AND FIO.iInVision = 6 THEN
        Lamp13_Green := TRUE;
END_IF		
IF nCounter = 13 AND FIO.iInVision = 9 THEN
        Lamp13_Metal := TRUE;
END_IF

//---------------------------------------------------

IF nCounter = 14 AND FIO.iInVision = 3 THEN
        Lamp14_Blue := TRUE;
END_IF	
IF nCounter = 14 AND FIO.iInVision = 6 THEN
        Lamp14_Green := TRUE;
END_IF		
IF nCounter = 14 AND FIO.iInVision = 9 THEN
        Lamp14_Metal := TRUE;
END_IF

//---------------------------------------------------

IF nCounter = 15 AND FIO.iInVision = 3 THEN
        Lamp15_Blue := TRUE;
END_IF	
IF nCounter = 15 AND FIO.iInVision = 6 THEN
        Lamp15_Green := TRUE;
END_IF		
IF nCounter = 15 AND FIO.iInVision = 9 THEN
        Lamp15_Metal := TRUE;
END_IF

//---------------------------------------------------

IF nCounter = 16 AND FIO.iInVision = 3 THEN
        Lamp16_Blue := TRUE;
END_IF	
IF nCounter = 16 AND FIO.iInVision = 6 THEN
        Lamp16_Green := TRUE;
END_IF		
IF nCounter = 16 AND FIO.iInVision = 9 THEN
        Lamp16_Metal := TRUE;
END_IF

//---------------------------------------------------

IF nCounter = 17 AND FIO.iInVision = 3 THEN
        Lamp17_Blue := TRUE;
END_IF	
IF nCounter = 17 AND FIO.iInVision = 6 THEN
        Lamp17_Green := TRUE;
END_IF		
IF nCounter = 17 AND FIO.iInVision = 9 THEN
        Lamp17_Metal := TRUE;
END_IF

//---------------------------------------------------

IF nCounter = 18 AND FIO.iInVision = 3 THEN
        Lamp18_Blue := TRUE;
END_IF	
IF nCounter = 18 AND FIO.iInVision = 6 THEN
        Lamp18_Green := TRUE;
END_IF		
IF nCounter = 18 AND FIO.iInVision = 9 THEN
        Lamp18_Metal := TRUE;
END_IF

//---------------------------------------------------

IF nCounter = 19 AND FIO.iInVision = 3 THEN
        Lamp19_Blue := TRUE;
END_IF	
IF nCounter = 19 AND FIO.iInVision = 6 THEN
        Lamp19_Green := TRUE;
END_IF		
IF nCounter = 19 AND FIO.iInVision = 9 THEN
        Lamp19_Metal := TRUE;
END_IF

//---------------------------------------------------

IF nCounter = 20 AND FIO.iInVision = 3 THEN
        Lamp20_Blue := TRUE;
END_IF	
IF nCounter = 20 AND FIO.iInVision = 6 THEN
        Lamp20_Green := TRUE;
END_IF		
IF nCounter = 20 AND FIO.iInVision = 9 THEN
        Lamp20_Metal := TRUE;
END_IF

//---------------------------------------------------

IF nCounter = 21 AND FIO.iInVision = 3 THEN
        Lamp21_Blue := TRUE;
END_IF	
IF nCounter = 21 AND FIO.iInVision = 6 THEN
        Lamp21_Green := TRUE;
END_IF		
IF nCounter = 21 AND FIO.iInVision = 9 THEN
        Lamp21_Metal := TRUE;
END_IF

//---------------------------------------------------

IF nCounter = 22 AND FIO.iInVision = 3 THEN
        Lamp22_Blue := TRUE;
END_IF	
IF nCounter = 22 AND FIO.iInVision = 6 THEN
        Lamp22_Green := TRUE;
END_IF		
IF nCounter = 22 AND FIO.iInVision = 9 THEN
        Lamp22_Metal := TRUE;
END_IF

//---------------------------------------------------

IF nCounter = 23 AND FIO.iInVision = 3 THEN
        Lamp23_Blue := TRUE;
END_IF	
IF nCounter = 23 AND FIO.iInVision = 6 THEN
        Lamp23_Green := TRUE;
END_IF		
IF nCounter = 23 AND FIO.iInVision = 9 THEN
        Lamp23_Metal := TRUE;
END_IF

//---------------------------------------------------

IF nCounter = 24 AND FIO.iInVision = 3 THEN
        Lamp24_Blue := TRUE;
END_IF	
IF nCounter = 24 AND FIO.iInVision = 6 THEN
        Lamp24_Green := TRUE;
END_IF		
IF nCounter = 24 AND FIO.iInVision = 9 THEN
        Lamp24_Metal := TRUE;
END_IF

//---------------------------------------------------

IF nCounter = 25 AND FIO.iInVision = 3 THEN
        Lamp25_Blue := TRUE;
END_IF	
IF nCounter = 25 AND FIO.iInVision = 6 THEN
        Lamp25_Green := TRUE;
END_IF		
IF nCounter = 25 AND FIO.iInVision = 9 THEN
        Lamp25_Metal := TRUE;
END_IF

//---------------------------------------------------

IF nCounter = 26 AND FIO.iInVision = 3 THEN
        Lamp26_Blue := TRUE;
END_IF	
IF nCounter = 26 AND FIO.iInVision = 6 THEN
        Lamp26_Green := TRUE;
END_IF		
IF nCounter = 26 AND FIO.iInVision = 9 THEN
        Lamp26_Metal := TRUE;
END_IF

//---------------------------------------------------

IF nCounter = 27 AND FIO.iInVision = 3 THEN
        Lamp27_Blue := TRUE;
END_IF	
IF nCounter = 27 AND FIO.iInVision = 6 THEN
        Lamp27_Green := TRUE;
END_IF		
IF nCounter = 27 AND FIO.iInVision = 9 THEN
        Lamp27_Metal := TRUE;
END_IF

//---------------------------------------------------

IF nCounter = 28 AND FIO.iInVision = 3 THEN
        Lamp28_Blue := TRUE;
END_IF	
IF nCounter = 28 AND FIO.iInVision = 6 THEN
        Lamp28_Green := TRUE;
END_IF		
IF nCounter = 28 AND FIO.iInVision = 9 THEN
        Lamp28_Metal := TRUE;
END_IF

//---------------------------------------------------

IF nCounter = 29 AND FIO.iInVision = 3 THEN
        Lamp29_Blue := TRUE;
END_IF	
IF nCounter = 29 AND FIO.iInVision = 6 THEN
        Lamp29_Green := TRUE;
END_IF		
IF nCounter = 29 AND FIO.iInVision = 9 THEN
        Lamp29_Metal := TRUE;
END_IF

//---------------------------------------------------

IF nCounter = 30 AND FIO.iInVision = 3 THEN
        Lamp30_Blue := TRUE;
END_IF	
IF nCounter = 30 AND FIO.iInVision = 6 THEN
        Lamp30_Green := TRUE;
END_IF		
IF nCounter = 30 AND FIO.iInVision = 9 THEN
        Lamp30_Metal := TRUE;
END_IF

//---------------------------------------------------

IF nCounter = 31 AND FIO.iInVision = 3 THEN
        Lamp31_Blue := TRUE;
END_IF	
IF nCounter = 31 AND FIO.iInVision = 6 THEN
        Lamp31_Green := TRUE;
END_IF		
IF nCounter = 31 AND FIO.iInVision = 9 THEN
        Lamp31_Metal := TRUE;
END_IF

//---------------------------------------------------

IF nCounter = 32 AND FIO.iInVision = 3 THEN
        Lamp32_Blue := TRUE;
END_IF	
IF nCounter = 32 AND FIO.iInVision = 6 THEN
        Lamp32_Green := TRUE;
END_IF		
IF nCounter = 32 AND FIO.iInVision = 9 THEN
        Lamp32_Metal := TRUE;
END_IF

//---------------------------------------------------

IF nCounter = 33 AND FIO.iInVision = 3 THEN
        Lamp33_Blue := TRUE;
END_IF	
IF nCounter = 33 AND FIO.iInVision = 6 THEN
        Lamp33_Green := TRUE;
END_IF		
IF nCounter = 33 AND FIO.iInVision = 9 THEN
        Lamp33_Metal := TRUE;
END_IF

//---------------------------------------------------

IF nCounter = 34 AND FIO.iInVision = 3 THEN
        Lamp34_Blue := TRUE;
END_IF	
IF nCounter = 34 AND FIO.iInVision = 6 THEN
        Lamp34_Green := TRUE;
END_IF		
IF nCounter = 34 AND FIO.iInVision = 9 THEN
        Lamp34_Metal := TRUE;
END_IF

//---------------------------------------------------

IF nCounter = 35 AND FIO.iInVision = 3 THEN
        Lamp35_Blue := TRUE;
END_IF	
IF nCounter = 35 AND FIO.iInVision = 6 THEN
        Lamp35_Green := TRUE;
END_IF		
IF nCounter = 35 AND FIO.iInVision = 9 THEN
        Lamp35_Metal := TRUE;
END_IF

//---------------------------------------------------

IF nCounter = 36 AND FIO.iInVision = 3 THEN
        Lamp36_Blue := TRUE;
END_IF	
IF nCounter = 36 AND FIO.iInVision = 6 THEN
        Lamp36_Green := TRUE;
END_IF		
IF nCounter = 36 AND FIO.iInVision = 9 THEN
        Lamp36_Metal := TRUE;
END_IF

//---------------------------------------------------

IF nCounter = 37 AND FIO.iInVision = 3 THEN
        Lamp37_Blue := TRUE;
END_IF	
IF nCounter = 37 AND FIO.iInVision = 6 THEN
        Lamp37_Green := TRUE;
END_IF		
IF nCounter = 37 AND FIO.iInVision = 9 THEN
        Lamp37_Metal := TRUE;
END_IF

//---------------------------------------------------

IF nCounter = 38 AND FIO.iInVision = 3 THEN
        Lamp38_Blue := TRUE;
END_IF	
IF nCounter = 38 AND FIO.iInVision = 6 THEN
        Lamp38_Green := TRUE;
END_IF		
IF nCounter = 38 AND FIO.iInVision = 9 THEN
        Lamp38_Metal := TRUE;
END_IF

//---------------------------------------------------

IF nCounter = 39 AND FIO.iInVision = 3 THEN
        Lamp39_Blue := TRUE;
END_IF	
IF nCounter = 39 AND FIO.iInVision = 6 THEN
        Lamp39_Green := TRUE;
END_IF		
IF nCounter = 39 AND FIO.iInVision = 9 THEN
        Lamp39_Metal := TRUE;
END_IF

//---------------------------------------------------

IF nCounter = 40 AND FIO.iInVision = 3 THEN
        Lamp40_Blue := TRUE;
END_IF	
IF nCounter = 40 AND FIO.iInVision = 6 THEN
        Lamp40_Green := TRUE;
END_IF		
IF nCounter = 40 AND FIO.iInVision = 9 THEN
        Lamp40_Metal := TRUE;
END_IF

//---------------------------------------------------

IF nCounter = 41 AND FIO.iInVision = 3 THEN
        Lamp41_Blue := TRUE;
END_IF	
IF nCounter = 41 AND FIO.iInVision = 6 THEN
        Lamp41_Green := TRUE;
END_IF		
IF nCounter = 41 AND FIO.iInVision = 9 THEN
        Lamp41_Metal := TRUE;
END_IF

//---------------------------------------------------

IF nCounter = 42 AND FIO.iInVision = 3 THEN
        Lamp42_Blue := TRUE;
END_IF	
IF nCounter = 42 AND FIO.iInVision = 6 THEN
        Lamp42_Green := TRUE;
END_IF		
IF nCounter = 42 AND FIO.iInVision = 9 THEN
        Lamp42_Metal := TRUE;
END_IF

//---------------------------------------------------

IF nCounter = 43 AND FIO.iInVision = 3 THEN
        Lamp43_Blue := TRUE;
END_IF	
IF nCounter = 43 AND FIO.iInVision = 6 THEN
        Lamp43_Green := TRUE;
END_IF		
IF nCounter = 43 AND FIO.iInVision = 9 THEN
        Lamp43_Metal := TRUE;
END_IF

//---------------------------------------------------

IF nCounter = 44 AND FIO.iInVision = 3 THEN
        Lamp44_Blue := TRUE;
END_IF	
IF nCounter = 44 AND FIO.iInVision = 6 THEN
        Lamp44_Green := TRUE;
END_IF		
IF nCounter = 44 AND FIO.iInVision = 9 THEN
        Lamp44_Metal := TRUE;
END_IF

//---------------------------------------------------

IF nCounter = 45 AND FIO.iInVision = 3 THEN
        Lamp45_Blue := TRUE;
END_IF	
IF nCounter = 45 AND FIO.iInVision = 6 THEN
        Lamp45_Green := TRUE;
END_IF		
IF nCounter = 45 AND FIO.iInVision = 9 THEN
        Lamp45_Metal := TRUE;
END_IF

//---------------------------------------------------

IF nCounter = 46 AND FIO.iInVision = 3 THEN
        Lamp46_Blue := TRUE;
END_IF	
IF nCounter = 46 AND FIO.iInVision = 6 THEN
        Lamp46_Green := TRUE;
END_IF		
IF nCounter = 46 AND FIO.iInVision = 9 THEN
        Lamp46_Metal := TRUE;
END_IF

//---------------------------------------------------

IF nCounter = 47 AND FIO.iInVision = 3 THEN
        Lamp47_Blue := TRUE;
END_IF	
IF nCounter = 47 AND FIO.iInVision = 6 THEN
        Lamp47_Green := TRUE;
END_IF		
IF nCounter = 47 AND FIO.iInVision = 9 THEN
        Lamp47_Metal := TRUE;
END_IF

//---------------------------------------------------

IF nCounter = 48 AND FIO.iInVision = 3 THEN
        Lamp48_Blue := TRUE;
END_IF	
IF nCounter = 48 AND FIO.iInVision = 6 THEN
        Lamp48_Green := TRUE;
END_IF		
IF nCounter = 48 AND FIO.iInVision = 9 THEN
        Lamp48_Metal := TRUE;
END_IF

//---------------------------------------------------

IF nCounter = 49 AND FIO.iInVision = 3 THEN
        Lamp49_Blue := TRUE;
END_IF	
IF nCounter = 49 AND FIO.iInVision = 6 THEN
        Lamp49_Green := TRUE;
END_IF		
IF nCounter = 49 AND FIO.iInVision = 9 THEN
        Lamp49_Metal := TRUE;
END_IF

//---------------------------------------------------

IF nCounter = 50 AND FIO.iInVision = 3 THEN
        Lamp50_Blue := TRUE;
END_IF	
IF nCounter = 50 AND FIO.iInVision = 6 THEN
        Lamp50_Green := TRUE;
END_IF		
IF nCounter = 50 AND FIO.iInVision = 9 THEN
        Lamp50_Metal := TRUE;
END_IF

//---------------------------------------------------

IF nCounter = 51 AND FIO.iInVision = 3 THEN
        Lamp41_Blue := TRUE;
END_IF	
IF nCounter = 51 AND FIO.iInVision = 6 THEN
        Lamp41_Green := TRUE;
END_IF		
IF nCounter = 51 AND FIO.iInVision = 9 THEN
        Lamp41_Metal := TRUE;
END_IF

//---------------------------------------------------

IF nCounter = 52 AND FIO.iInVision = 3 THEN
        Lamp52_Blue := TRUE;
END_IF	
IF nCounter = 52 AND FIO.iInVision = 6 THEN
        Lamp52_Green := TRUE;
END_IF		
IF nCounter = 52 AND FIO.iInVision = 9 THEN
        Lamp52_Metal := TRUE;
END_IF

//---------------------------------------------------

IF nCounter = 53 AND FIO.iInVision = 3 THEN
        Lamp53_Blue := TRUE;
END_IF	
IF nCounter = 53 AND FIO.iInVision = 6 THEN
        Lamp53_Green := TRUE;
END_IF		
IF nCounter = 53 AND FIO.iInVision = 9 THEN
        Lamp53_Metal := TRUE;
END_IF

//---------------------------------------------------

IF nCounter = 54 AND FIO.iInVision = 3 THEN
        Lamp54_Blue := TRUE;
END_IF	
IF nCounter = 54 AND FIO.iInVision = 6 THEN
        Lamp54_Green := TRUE;
END_IF		
IF nCounter = 54 AND FIO.iInVision = 9 THEN
        Lamp54_Metal := TRUE;
END_IF

//---------------------------------------------------

END_PROGRAM

// ---- GlobalTextList.TcGTLO
TEXTLIST GlobalTextList
  567 = '%f'
  696 = '%f0.2'
  761 = 'COUNTER'
  472 = 'Plads: 1'
  850 = 'Plads: 10'
  785 = 'Plads: 11'
  364 = 'Plads: 12'
  894 = 'Plads: 13'
  898 = 'Plads: 14'
  84 = 'Plads: 15'
  18 = 'Plads: 16'
  810 = 'Plads: 17'
  989 = 'Plads: 18'
  722 = 'Plads: 19'
  120 = 'Plads: 2'
  566 = 'Plads: 20'
  543 = 'Plads: 21'
  8 = 'Plads: 22'
  479 = 'Plads: 23'
  745 = 'Plads: 24'
  889 = 'Plads: 25'
  19 = 'Plads: 26'
  498 = 'Plads: 27'
  359 = 'Plads: 28'
  792 = 'Plads: 29'
  313 = 'Plads: 3'
  759 = 'Plads: 30'
  795 = 'Plads: 31'
  385 = 'Plads: 32'
  648 = 'Plads: 33'
  131 = 'Plads: 34'
  923 = 'Plads: 35'
  565 = 'Plads: 36'
  62 = 'Plads: 37'
  422 = 'Plads: 38'
  344 = 'Plads: 39'
  248 = 'Plads: 4'
  195 = 'Plads: 40'
  779 = 'Plads: 41'
  914 = 'Plads: 42'
  345 = 'Plads: 43'
  791 = 'Plads: 44'
  806 = 'Plads: 45'
  246 = 'Plads: 46'
  840 = 'Plads: 47'
  695 = 'Plads: 48'
  999 = 'Plads: 49'
  71 = 'Plads: 5'
  272 = 'Plads: 50'
  622 = 'Plads: 51'
  717 = 'Plads: 52'
  603 = 'Plads: 53'
  138 = 'Plads: 54'
  271 = 'Plads: 6'
  920 = 'Plads: 7'
  868 = 'Plads: 8'
  284 = 'Plads: 9'
  1178 = 'RESET'
  488 = 'START'
  285 = 'STATUS'
  121 = 'STOP'
END_TEXTLIST

// ---- VISUs/Visualization_Pos.TcVIS
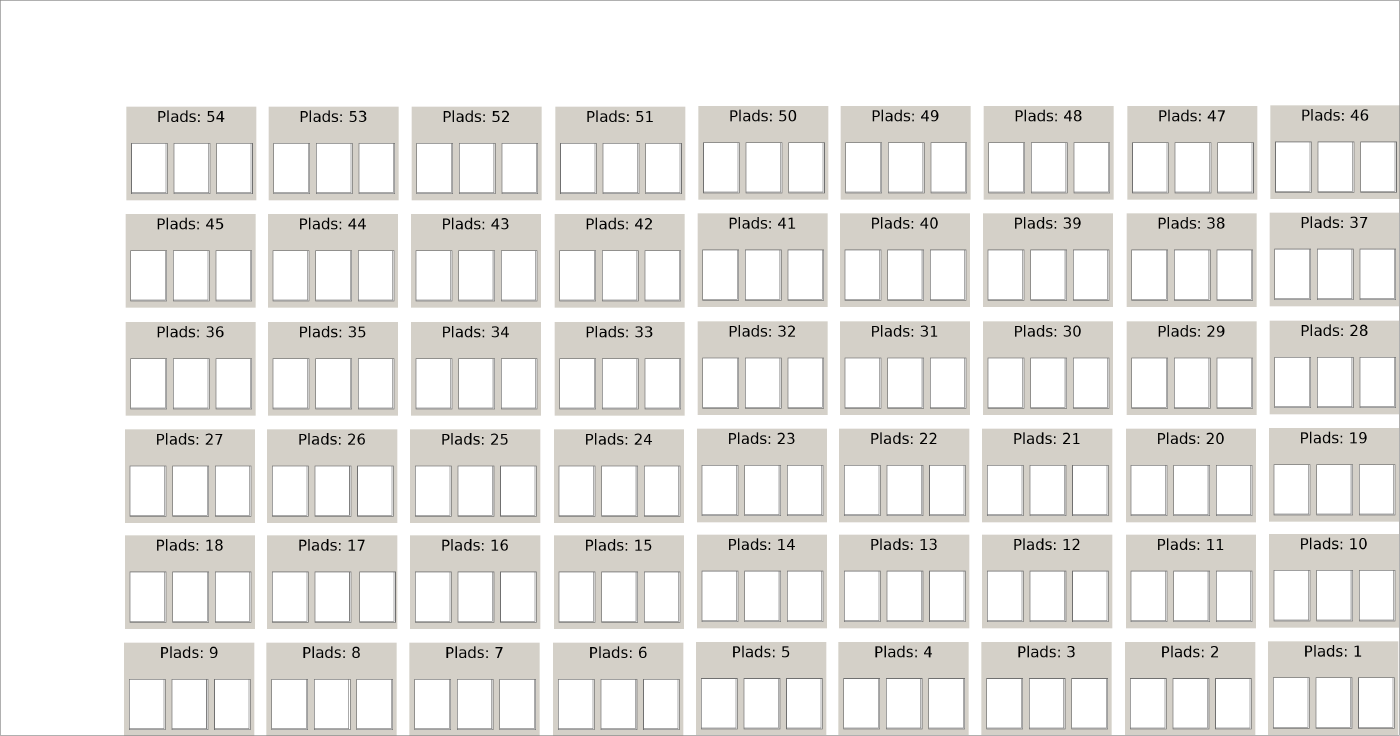
VISUALIZATION Visualization_Pos  // 2007x1056
    Textfield (1818,920 186x134), "Plads: 1", colour toggle: MAIN.Occ
    Button (1886,972 52x73), colour toggle: HMI.Lamp1_Green
        toggle HMI.Lamp1_Green
    Button (1825,972 52x73), colour toggle: HMI.Lamp1_Metal
    Button (1947,972 52x73), colour toggle: HMI.Lamp1_Blue
        toggle HMI.Lamp1_Blue
    Textfield (1613,921 186x134), "Plads: 2", colour toggle: MAIN.Occ
    Button (1681,973 52x73), colour toggle: HMI.Lamp2_Green
    Button (1620,973 52x73)
    Button (1742,973 52x73), colour toggle: HMI.Lamp2_Blue
    Textfield (1407,921 186x134), "Plads: 3", colour toggle: MAIN.Occ
    Button (1475,973 52x73), colour toggle: HMI.Lamp3_Green
    Button (1414,973 52x73), colour toggle: HMI.Lamp3_Metal
    Button (1536,973 52x73), colour toggle: HMI.Lamp3_Blue
    Textfield (1202,921 186x134), "Plads: 4"
    Button (1270,973 52x73), colour toggle: HMI.Lamp4_Green
    Button (1209,973 52x73), colour toggle: HMI.Lamp4_Metal
    Button (1331,973 52x73), colour toggle: HMI.Lamp4_Blue
    Textfield (998,921 186x134), "Plads: 5"
    Button (1066,973 52x73)
    Button (1005,973 52x73)
    Button (1127,973 52x73), colour toggle: MAIN.bStart
    Textfield (793,922 186x134), "Plads: 6"
    Button (861,974 52x73), colour toggle: HMI.Lamp6_Green
    Button (800,974 52x73), colour toggle: HMI.Lamp6_Metal
    Button (922,974 52x73), colour toggle: HMI.Lamp6_Blue
    Textfield (587,922 186x134), "Plads: 7"
    Button (655,974 52x73), colour toggle: HMI.Lamp7_Green
    Button (594,974 52x73), colour toggle: HMI.Lamp7_Metal
    Button (716,974 52x73), colour toggle: HMI.Lamp7_Blue
    Textfield (382,922 186x134), "Plads: 8"
    Button (450,974 52x73), colour toggle: HMI.Lamp8_Green
    Button (389,974 52x73), colour toggle: HMI.Lamp8_Metal
    Button (511,974 52x73), colour toggle: HMI.Lamp8_Blue
    Textfield (178,922 186x134), "Plads: 9"
    Button (246,974 52x73), colour toggle: HMI.Lamp9_Green
    Button (185,974 52x73), colour toggle: HMI.Lamp9_Metal
    Button (307,974 52x73), colour toggle: HMI.Lamp9_Blue
    Textfield (1819,766 186x134), "Plads: 10"
    Button (1887,818 52x73), colour toggle: HMI.Lamp10_Green
    Button (1826,818 52x73), colour toggle: HMI.Lamp10_Metal
    Button (1948,818 52x73), colour toggle: HMI.Lamp10_Blue
    Textfield (1614,767 186x134), "Plads: 11"
    Button (1682,819 52x73), colour toggle: HMI.Lamp11_Green
    Button (1621,819 52x73), colour toggle: HMI.Lamp11_Metal
    Button (1743,819 52x73), colour toggle: HMI.Lamp11_Blue
    Textfield (1408,767 186x134), "Plads: 12"
    Button (1476,819 52x73), colour toggle: HMI.Lamp12_Green
    Button (1415,819 52x73), colour toggle: HMI.Lamp12_Metal
    Button (1537,819 52x73), colour toggle: HMI.Lamp12_Blue
    Textfield (1203,767 186x134), "Plads: 13"
    Button (1271,819 52x73), colour toggle: HMI.Lamp13_Green
    Button (1210,819 52x73), colour toggle: HMI.Lamp13_Metal
    Button (1332,819 52x73), colour toggle: HMI.Lamp13_Blue
    Textfield (999,767 186x134), "Plads: 14"
    Button (1067,819 52x73), colour toggle: HMI.Lamp14_Green
    Button (1006,819 52x73), colour toggle: HMI.Lamp14_Metal
    Button (1128,819 52x73), colour toggle: HMI.Lamp14_Blue
    Textfield (794,768 186x134), "Plads: 15"
    Button (862,820 52x73), colour toggle: HMI.Lamp15_Green
    Button (801,820 52x73), colour toggle: HMI.Lamp15_Metal
    Button (923,820 52x73), colour toggle: HMI.Lamp15_Blue
    Textfield (588,768 186x134), "Plads: 16"
    Button (656,820 52x73), colour toggle: HMI.Lamp16_Green
    Button (595,820 52x73), colour toggle: HMI.Lamp16_Metal
    Button (717,820 52x73), colour toggle: HMI.Lamp16_Blue
    Textfield (383,768 186x134), "Plads: 17"
    Button (451,820 52x73), colour toggle: HMI.Lamp17_Green
    Button (390,820 52x73), colour toggle: HMI.Lamp17_Metal
    Button (515,820 52x73), colour toggle: HMI.Lamp17_Blue
    Textfield (179,768 186x134), "Plads: 18"
    Button (247,820 52x73), colour toggle: HMI.Lamp18_Green
    Button (186,820 52x73), colour toggle: HMI.Lamp18_Metal
    Button (308,820 52x73), colour toggle: HMI.Lamp18_Blue
    Textfield (1819,614 186x134), "Plads: 19"
    Button (1887,666 52x73), colour toggle: HMI.Lamp19_Green
    Button (1826,666 52x73), colour toggle: HMI.Lamp19_Metal
    Button (1948,666 52x73), colour toggle: HMI.Lamp19_Blue
    Textfield (1614,615 186x134), "Plads: 20"
    Button (1682,667 52x73), colour toggle: HMI.Lamp20_Green
    Button (1621,667 52x73), colour toggle: HMI.Lamp20_Metal
    Button (1743,667 52x73), colour toggle: HMI.Lamp20_Blue
    Textfield (1408,615 186x134), "Plads: 21"
    Button (1476,667 52x73), colour toggle: HMI.Lamp21_Green
    Button (1415,667 52x73), colour toggle: HMI.Lamp21_Metal
    Button (1537,667 52x73), colour toggle: HMI.Lamp21_Blue
    Textfield (1203,615 186x134), "Plads: 22"
    Button (1271,667 52x73), colour toggle: HMI.Lamp22_Green
    Button (1210,667 52x73), colour toggle: HMI.Lamp22_Metal
    Button (1332,667 52x73), colour toggle: HMI.Lamp22_Blue
    Textfield (999,615 186x134), "Plads: 23"
    Button (1067,667 52x73), colour toggle: HMI.Lamp23_Green
    Button (1006,667 52x73), colour toggle: HMI.Lamp23_Metal
    Button (1128,667 52x73), colour toggle: HMI.Lamp23_Blue
    Textfield (794,616 186x134), "Plads: 24"
    Button (862,668 52x73), colour toggle: HMI.Lamp24_Green
    Button (801,668 52x73), colour toggle: HMI.Lamp24_Metal
    Button (923,668 52x73), colour toggle: HMI.Lamp24_Blue
    Textfield (588,616 186x134), "Plads: 25"
    Button (656,668 52x73), colour toggle: HMI.Lamp25_Green
    Button (595,668 52x73), colour toggle: HMI.Lamp25_Metal
    Button (717,668 52x73), colour toggle: HMI.Lamp25_Blue
    Textfield (383,616 186x134), "Plads: 26"
    Button (451,668 52x73), colour toggle: HMI.Lamp26_Green
    Button (390,668 52x73), colour toggle: HMI.Lamp26_Metal
    Button (512,668 52x73), colour toggle: HMI.Lamp26_Blue
    Textfield (179,616 186x134), "Plads: 27"
    Button (247,668 52x73), colour toggle: HMI.Lamp27_Green
    Button (186,668 52x73), colour toggle: HMI.Lamp27_Metal
    Button (308,668 52x73), colour toggle: HMI.Lamp27_Blue
    Textfield (1820,460 186x134), "Plads: 28"
    Button (1888,512 52x73), colour toggle: HMI.Lamp28_Green
    Button (1827,512 52x73), colour toggle: HMI.Lamp28_Metal
    Button (1949,512 52x73), colour toggle: HMI.Lamp28_Blue
    Textfield (1615,461 186x134), "Plads: 29"
    Button (1683,513 52x73), colour toggle: HMI.Lamp29_Green
    Button (1622,513 52x73), colour toggle: HMI.Lamp29_Metal
    Button (1744,513 52x73), colour toggle: HMI.Lamp29_Blue
    Textfield (1409,461 186x134), "Plads: 30"
    Button (1477,513 52x73), colour toggle: HMI.Lamp30_Green
    Button (1416,513 52x73), colour toggle: HMI.Lamp30_Metal
    Button (1538,513 52x73), colour toggle: HMI.Lamp30_Blue
    Textfield (1204,461 186x134), "Plads: 31"
    Button (1272,513 52x73), colour toggle: HMI.Lamp31_Green
    Button (1211,513 52x73), colour toggle: HMI.Lamp31_Metal
    Button (1333,513 52x73), colour toggle: HMI.Lamp31_Blue
    Textfield (1000,461 186x134), "Plads: 32"
    Button (1068,513 52x73), colour toggle: HMI.Lamp32_Green
    Button (1007,513 52x73), colour toggle: HMI.Lamp32_Metal
    Button (1129,513 52x73), colour toggle: HMI.Lamp32_Blue
    Textfield (795,462 186x134), "Plads: 33"
    Button (863,514 52x73), colour toggle: HMI.Lamp33_Green
    Button (802,514 52x73), colour toggle: HMI.Lamp33_Metal
    Button (924,514 52x73), colour toggle: HMI.Lamp33_Blue
    Textfield (589,462 186x134), "Plads: 34"
    Button (657,514 52x73), colour toggle: HMI.Lamp34_Blue
    Button (596,514 52x73), colour toggle: HMI.Lamp34_Metal
    Button (718,514 52x73), colour toggle: HMI.Lamp34_Blue
    Textfield (384,462 186x134), "Plads: 35"
    Button (452,514 52x73), colour toggle: HMI.Lamp35_Green
    Button (391,514 52x73), colour toggle: HMI.Lamp35_Metal
    Button (513,514 52x73), colour toggle: HMI.Lamp35_Blue
    Textfield (180,462 186x134), "Plads: 36"
    Button (248,514 52x73), colour toggle: HMI.Lamp36_Green
    Button (187,514 52x73), colour toggle: HMI.Lamp36_Metal
    Button (309,514 52x73), colour toggle: HMI.Lamp36_Blue
    Textfield (1820,305 186x134), "Plads: 37"
    Button (1888,357 52x73), colour toggle: HMI.Lamp37_Green
    Button (1827,357 52x73), colour toggle: HMI.Lamp37_Metal
    Button (1949,357 52x73), colour toggle: HMI.Lamp37_Blue
    Textfield (1615,306 186x134), "Plads: 38"
    Button (1683,358 52x73), colour toggle: HMI.Lamp38_Green
    Button (1622,358 52x73), colour toggle: HMI.Lamp38_Metal
    Button (1744,358 52x73), colour toggle: HMI.Lamp38_Blue
    Textfield (1409,306 186x134), "Plads: 39"
    Button (1477,358 52x73), colour toggle: HMI.Lamp39_Green
    Button (1416,358 52x73), colour toggle: HMI.Lamp39_Metal
    Button (1538,358 52x73), colour toggle: HMI.Lamp39_Blue
    Textfield (1204,306 186x134), "Plads: 40"
    Button (1272,358 52x73), colour toggle: HMI.Lamp40_Green
    Button (1211,358 52x73), colour toggle: HMI.Lamp40_Metal
    Button (1333,358 52x73), colour toggle: HMI.Lamp40_Blue
    Textfield (1000,306 186x134), "Plads: 41"
    Button (1068,358 52x73), colour toggle: HMI.Lamp41_Green
    Button (1007,358 52x73), colour toggle: HMI.Lamp41_Metal
    Button (1129,358 52x73), colour toggle: HMI.Lamp41_Blue
    Textfield (795,307 186x134), "Plads: 42"
    Button (863,359 52x73), colour toggle: HMI.Lamp42_Green
    Button (802,359 52x73), colour toggle: HMI.Lamp42_Metal
    Button (924,359 52x73), colour toggle: HMI.Lamp42_Blue
    Textfield (589,307 186x134), "Plads: 43"
    Button (657,359 52x73), colour toggle: HMI.Lamp43_Green
    Button (596,359 52x73), colour toggle: HMI.Lamp43_Metal
    Button (718,359 52x73), colour toggle: HMI.Lamp43_Blue
    Textfield (384,307 186x134), "Plads: 44"
    Button (452,359 52x73), colour toggle: HMI.Lamp44_Green
    Button (391,359 52x73), colour toggle: HMI.Lamp44_Metal
    Button (513,359 52x73), colour toggle: HMI.Lamp44_Blue
    Textfield (180,307 186x134), "Plads: 45"
    Button (248,359 52x73), colour toggle: HMI.Lamp45_Green
    Button (187,359 52x73), colour toggle: HMI.Lamp45_Metal
    Button (309,359 52x73), colour toggle: HMI.Lamp45_Blue
    Textfield (1821,151 186x134), "Plads: 46"
    Button (1889,203 52x73), colour toggle: HMI.Lamp46_Green
    Button (1828,203 52x73), colour toggle: HMI.Lamp46_Metal
    Button (1950,203 52x73), colour toggle: HMI.Lamp46_Blue
    Textfield (1616,152 186x134), "Plads: 47"
    Button (1684,204 52x73), colour toggle: HMI.Lamp47_Green
    Button (1623,204 52x73), colour toggle: HMI.Lamp47_Metal
    Button (1745,204 52x73), colour toggle: HMI.Lamp47_Blue
    Textfield (1410,152 186x134), "Plads: 48"
    Button (1478,204 52x73), colour toggle: HMI.Lamp48_Green
    Button (1417,204 52x73), colour toggle: HMI.Lamp48_Metal
    Button (1539,204 52x73), colour toggle: HMI.Lamp48_Blue
    Textfield (1205,152 186x134), "Plads: 49"
    Button (1273,204 52x73), colour toggle: HMI.Lamp49_Green
    Button (1212,204 52x73), colour toggle: HMI.Lamp49_Metal
    Button (1334,204 52x73), colour toggle: HMI.Lamp49_Blue
    Textfield (1001,152 186x134), "Plads: 50"
    Button (1069,204 52x73), colour toggle: HMI.Lamp50_Green
    Button (1008,204 52x73), colour toggle: HMI.Lamp50_Metal
    Button (1130,204 52x73), colour toggle: HMI.Lamp50_Blue
    Textfield (796,153 186x134), "Plads: 51"
    Button (864,205 52x73), colour toggle: HMI.Lamp51_Green
    Button (803,205 52x73), colour toggle: HMI.Lamp51_Metal
    Button (925,205 52x73), colour toggle: HMI.Lamp51_Blue
    Textfield (590,153 186x134), "Plads: 52"
    Button (658,205 52x73), colour toggle: HMI.Lamp52_Green
    Button (597,205 52x73), colour toggle: HMI.Lamp52_Metal
    Button (719,205 52x73), colour toggle: HMI.Lamp52_Blue
    Textfield (385,153 186x134), "Plads: 53"
    Button (453,205 52x73), colour toggle: HMI.Lamp53_Green
    Button (392,205 52x73), colour toggle: HMI.Lamp53_Metal
    Button (514,205 52x73), colour toggle: HMI.Lamp53_Blue
    Textfield (181,153 186x134), "Plads: 54"
    Button (249,205 52x73), colour toggle: HMI.Lamp54_Green
    Button (188,205 52x73), colour toggle: HMI.Lamp54_Metal
    Button (310,205 52x73), colour toggle: HMI.Lamp54_Blue
END_VISUALIZATION

// ---- VISUs/Visualization_Start_Screen.TcVIS
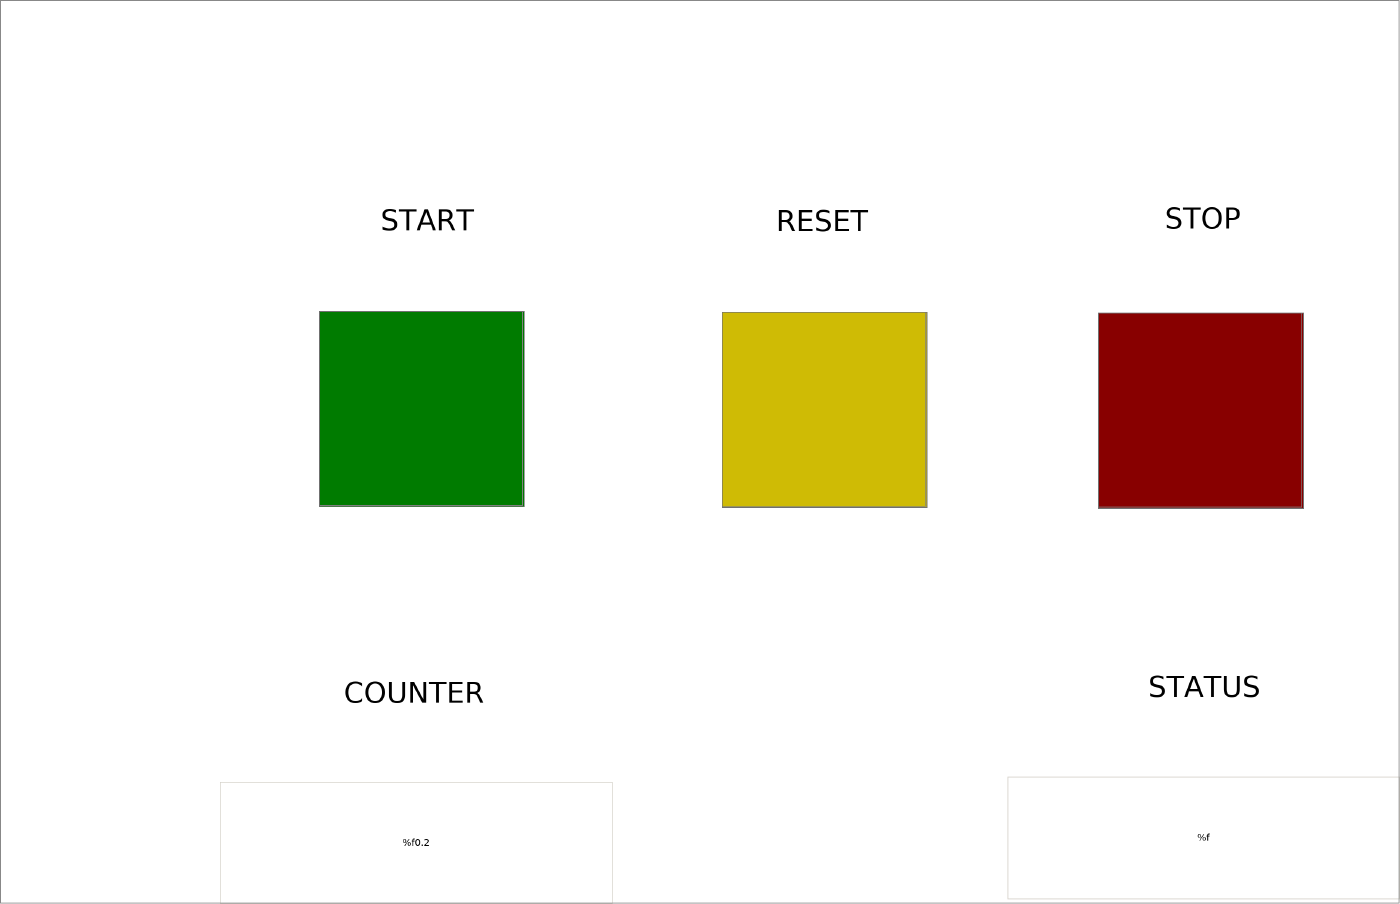
VISUALIZATION Visualization_Start_Screen  // 1637x1058
    Button (373,364 240x229), colour toggle: FIO.bEbStart
        OnMouseClick: toggle FIO.bEbStart
    Button (1284,366 240x229), colour toggle: FIO.bEbStopLight
        toggle FIO.bEbStop
        OnMouseClick: toggle FIO.bEbStop
    Textfield (257,915 459x143), "%f0.2", text variable: FIO.iEbCounter
    Textfield (1178,909 459x143), "%f", text variable: FIO.bEbAuto
    Textfield (399,230 201x55), "START"
    Textfield (1306,228 201x55), "STOP"
    Textfield (384,783 201x55), "COUNTER"
    Textfield (1308,776 201x55), "STATUS"
    Button (844,365 240x229), colour toggle: FIO.bEbReset
        OnMouseClick: toggle FIO.bEbReset
    Textfield (861,231 201x55), "RESET"
END_VISUALIZATION
